// TIA Portal V20 export
FUNCTION "01 T5 EXCENTRIC Alarms" : Void   // FC1118, LAD
TITLE = ALARMS
{ S7_Optimized_Access := 'TRUE' }
// stored: AutoNumber false, IsIECCheckEnabled true, SetENOAutomatically false
   VAR_TEMP
      Trash : Bool;
   END_VAR
BEGIN

REGION Network 1: ============ ALARMS RESET ============
END_REGION

REGION Network 2: Alarms Reset
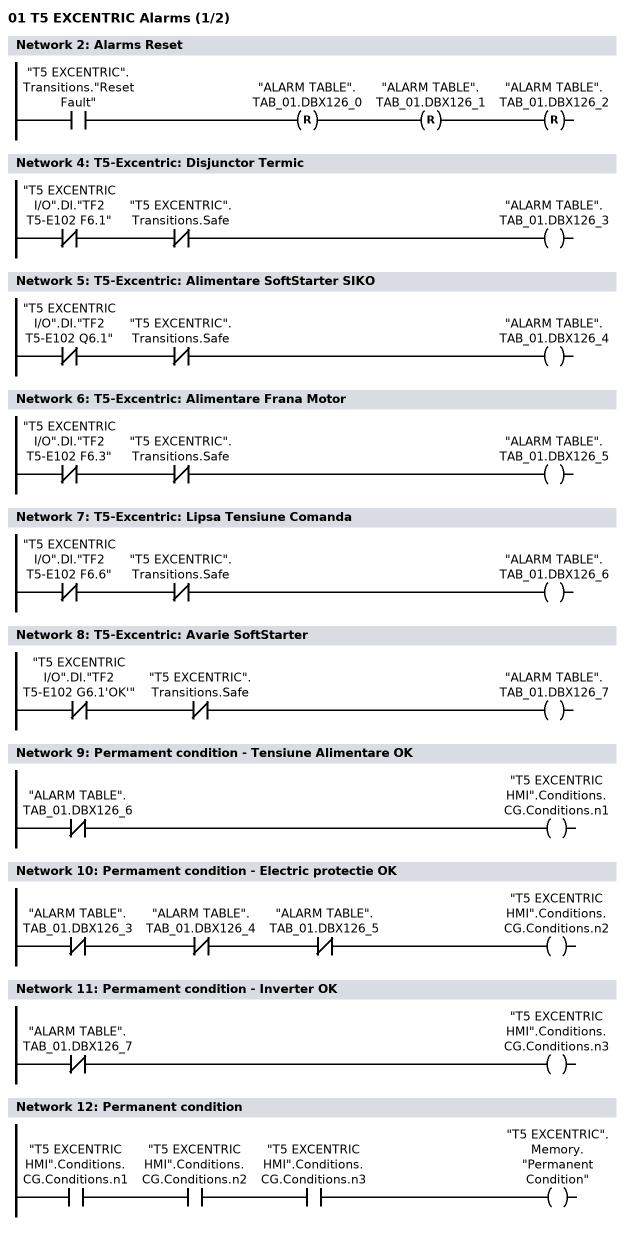
   RUNG wire#powerrail
      Contact( "T5 EXCENTRIC".Transitions."Reset Fault" )
      R_Coil( "ALARM TABLE".TAB_01.DBX126_0 )
      R_Coil( "ALARM TABLE".TAB_01.DBX126_1 )
      R_Coil( "ALARM TABLE".TAB_01.DBX126_2 )
   END_RUNG
   // the same network as SCL:
   IF "T5 EXCENTRIC".Transitions."Reset Fault" THEN
       "ALARM TABLE".TAB_01.DBX126_0 := FALSE;
       "ALARM TABLE".TAB_01.DBX126_1 := FALSE;
       "ALARM TABLE".TAB_01.DBX126_2 := FALSE;
   END_IF;
END_REGION

REGION Network 3: ============ PERMANENT CONDITIONS ============
END_REGION

REGION Network 4: T5-Excentric: Disjunctor Termic
   RUNG wire#powerrail
      I_Contact( "T5 EXCENTRIC I/O".DI."TF2 T5-E102 F6.1" )
      I_Contact( "T5 EXCENTRIC".Transitions.Safe )
      Coil( "ALARM TABLE".TAB_01.DBX126_3 )
   END_RUNG
   // the same network as SCL:
   "ALARM TABLE".TAB_01.DBX126_3 := NOT "T5 EXCENTRIC I/O".DI."TF2 T5-E102 F6.1" AND NOT "T5 EXCENTRIC".Transitions.Safe;
END_REGION

REGION Network 5: T5-Excentric: Alimentare SoftStarter SIKO
   RUNG wire#powerrail
      I_Contact( "T5 EXCENTRIC I/O".DI."TF2 T5-E102 Q6.1" )
      I_Contact( "T5 EXCENTRIC".Transitions.Safe )
      Coil( "ALARM TABLE".TAB_01.DBX126_4 )
   END_RUNG
   // the same network as SCL:
   "ALARM TABLE".TAB_01.DBX126_4 := NOT "T5 EXCENTRIC I/O".DI."TF2 T5-E102 Q6.1" AND NOT "T5 EXCENTRIC".Transitions.Safe;
END_REGION

REGION Network 6: T5-Excentric: Alimentare Frana Motor
   RUNG wire#powerrail
      I_Contact( "T5 EXCENTRIC I/O".DI."TF2 T5-E102 F6.3" )
      I_Contact( "T5 EXCENTRIC".Transitions.Safe )
      Coil( "ALARM TABLE".TAB_01.DBX126_5 )
   END_RUNG
   // the same network as SCL:
   "ALARM TABLE".TAB_01.DBX126_5 := NOT "T5 EXCENTRIC I/O".DI."TF2 T5-E102 F6.3" AND NOT "T5 EXCENTRIC".Transitions.Safe;
END_REGION

REGION Network 7: T5-Excentric: Lipsa Tensiune Comanda
   RUNG wire#powerrail
      I_Contact( "T5 EXCENTRIC I/O".DI."TF2 T5-E102 F6.6" )
      I_Contact( "T5 EXCENTRIC".Transitions.Safe )
      Coil( "ALARM TABLE".TAB_01.DBX126_6 )
   END_RUNG
   // the same network as SCL:
   "ALARM TABLE".TAB_01.DBX126_6 := NOT "T5 EXCENTRIC I/O".DI."TF2 T5-E102 F6.6" AND NOT "T5 EXCENTRIC".Transitions.Safe;
END_REGION

REGION Network 8: T5-Excentric: Avarie SoftStarter
   RUNG wire#powerrail
      I_Contact( "T5 EXCENTRIC I/O".DI."TF2 T5-E102 G6.1'OK'" )
      I_Contact( "T5 EXCENTRIC".Transitions.Safe )
      Coil( "ALARM TABLE".TAB_01.DBX126_7 )
   END_RUNG
   // the same network as SCL:
   "ALARM TABLE".TAB_01.DBX126_7 := NOT "T5 EXCENTRIC I/O".DI."TF2 T5-E102 G6.1'OK'" AND NOT "T5 EXCENTRIC".Transitions.Safe;
END_REGION

REGION Network 9: Permament condition - Tensiune Alimentare OK
   RUNG wire#powerrail
      I_Contact( "ALARM TABLE".TAB_01.DBX126_6 )
      Coil( "T5 EXCENTRIC HMI".Conditions.CG.Conditions.n1 )
   END_RUNG
   // the same network as SCL:
   "T5 EXCENTRIC HMI".Conditions.CG.Conditions.n1 := NOT "ALARM TABLE".TAB_01.DBX126_6;
END_REGION

REGION Network 10: Permament condition - Electric protectie OK
   RUNG wire#powerrail
      I_Contact( "ALARM TABLE".TAB_01.DBX126_3 )
      I_Contact( "ALARM TABLE".TAB_01.DBX126_4 )
      I_Contact( "ALARM TABLE".TAB_01.DBX126_5 )
      Coil( "T5 EXCENTRIC HMI".Conditions.CG.Conditions.n2 )
   END_RUNG
   // the same network as SCL:
   "T5 EXCENTRIC HMI".Conditions.CG.Conditions.n2 := NOT "ALARM TABLE".TAB_01.DBX126_3 AND NOT "ALARM TABLE".TAB_01.DBX126_4 AND NOT "ALARM TABLE".TAB_01.DBX126_5;
END_REGION

REGION Network 11: Permament condition - Inverter OK
   RUNG wire#powerrail
      I_Contact( "ALARM TABLE".TAB_01.DBX126_7 )
      Coil( "T5 EXCENTRIC HMI".Conditions.CG.Conditions.n3 )
   END_RUNG
   // the same network as SCL:
   "T5 EXCENTRIC HMI".Conditions.CG.Conditions.n3 := NOT "ALARM TABLE".TAB_01.DBX126_7;
END_REGION

REGION Network 12: Permanent condition
   RUNG wire#powerrail
      Contact( "T5 EXCENTRIC HMI".Conditions.CG.Conditions.n1 )
      Contact( "T5 EXCENTRIC HMI".Conditions.CG.Conditions.n2 )
      Contact( "T5 EXCENTRIC HMI".Conditions.CG.Conditions.n3 )
      Coil( "T5 EXCENTRIC".Memory."Permanent Condition" )
   END_RUNG
   // the same network as SCL:
   "T5 EXCENTRIC".Memory."Permanent Condition" := "T5 EXCENTRIC HMI".Conditions.CG.Conditions.n1 AND "T5 EXCENTRIC HMI".Conditions.CG.Conditions.n2 AND "T5 EXCENTRIC HMI".Conditions.CG.Conditions.n3;
END_REGION

REGION Network 13: ======= MACHINE MOVEMENT CONTROL (SENSORS / ENCODERS / INTERLOCKS) =======
END_REGION

REGION Network 14: T5-Excentric: TimeOut Deplasare 'Inainte'
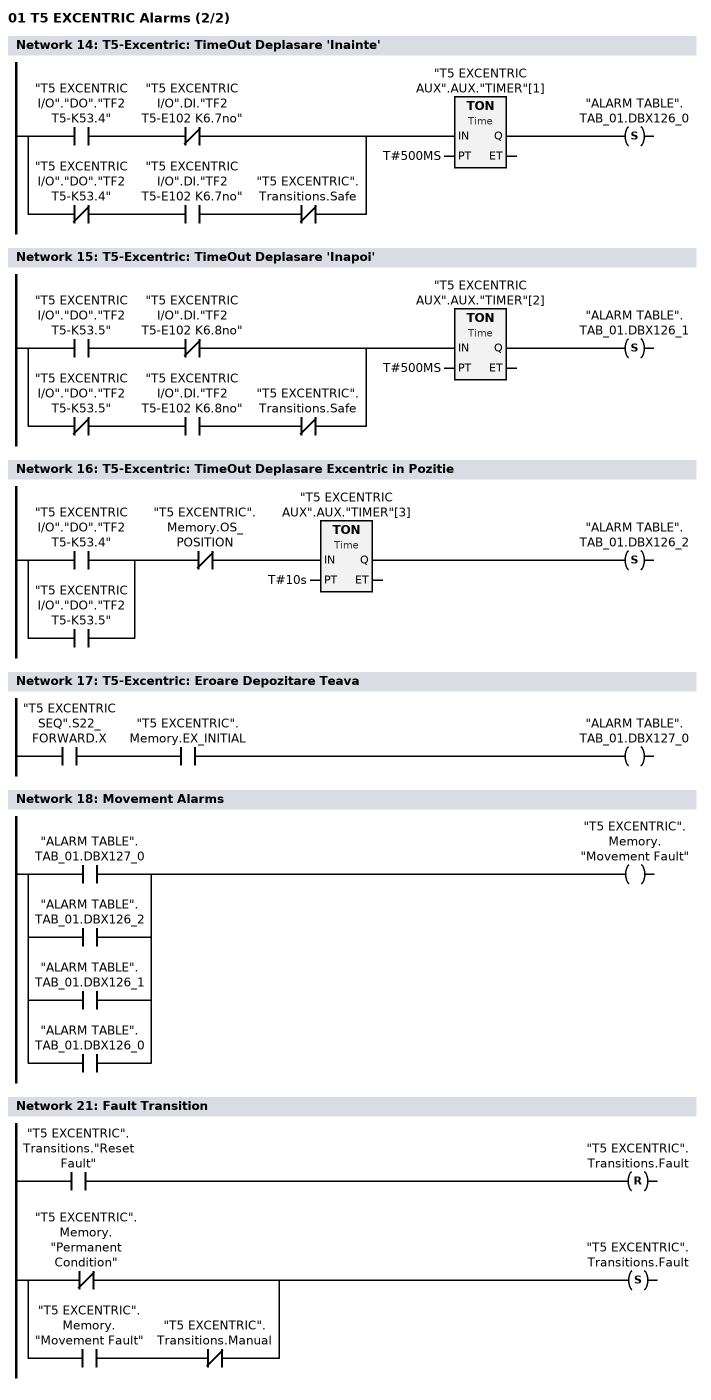
   RUNG wire#powerrail
      Contact( "T5 EXCENTRIC I/O"."DO"."TF2 T5-K53.4" )
      I_Contact( "T5 EXCENTRIC I/O".DI."TF2 T5-E102 K6.7no" )
      wire#w1
      { S7_Templates := "time_type := Time" } "T5 EXCENTRIC AUX".AUX."TIMER"[1].TON(pt := T#500MS, et =>)
      S_Coil( "ALARM TABLE".TAB_01.DBX126_0 )
   END_RUNG
   RUNG wire#powerrail
      I_Contact( "T5 EXCENTRIC I/O"."DO"."TF2 T5-K53.4" )
      Contact( "T5 EXCENTRIC I/O".DI."TF2 T5-E102 K6.7no" )
      I_Contact( "T5 EXCENTRIC".Transitions.Safe )
   END_RUNG wire#w1
   // the same network as SCL:
   "T5 EXCENTRIC AUX".AUX."TIMER"[1].TON(IN := ("T5 EXCENTRIC I/O"."DO"."TF2 T5-K53.4" AND NOT "T5 EXCENTRIC I/O".DI."TF2 T5-E102 K6.7no") OR (NOT "T5 EXCENTRIC I/O"."DO"."TF2 T5-K53.4" AND "T5 EXCENTRIC I/O".DI."TF2 T5-E102 K6.7no" AND NOT "T5 EXCENTRIC".Transitions.Safe),
                           PT := T#500MS);
   IF "T5 EXCENTRIC AUX".AUX."TIMER"[1].Q THEN "ALARM TABLE".TAB_01.DBX126_0 := TRUE; END_IF;
END_REGION

REGION Network 15: T5-Excentric: TimeOut Deplasare 'Inapoi'
   RUNG wire#powerrail
      Contact( "T5 EXCENTRIC I/O"."DO"."TF2 T5-K53.5" )
      I_Contact( "T5 EXCENTRIC I/O".DI."TF2 T5-E102 K6.8no" )
      wire#w1
      { S7_Templates := "time_type := Time" } "T5 EXCENTRIC AUX".AUX."TIMER"[2].TON(pt := T#500MS, et =>)
      S_Coil( "ALARM TABLE".TAB_01.DBX126_1 )
   END_RUNG
   RUNG wire#powerrail
      I_Contact( "T5 EXCENTRIC I/O"."DO"."TF2 T5-K53.5" )
      Contact( "T5 EXCENTRIC I/O".DI."TF2 T5-E102 K6.8no" )
      I_Contact( "T5 EXCENTRIC".Transitions.Safe )
   END_RUNG wire#w1
   // the same network as SCL:
   "T5 EXCENTRIC AUX".AUX."TIMER"[2].TON(IN := ("T5 EXCENTRIC I/O"."DO"."TF2 T5-K53.5" AND NOT "T5 EXCENTRIC I/O".DI."TF2 T5-E102 K6.8no") OR (NOT "T5 EXCENTRIC I/O"."DO"."TF2 T5-K53.5" AND "T5 EXCENTRIC I/O".DI."TF2 T5-E102 K6.8no" AND NOT "T5 EXCENTRIC".Transitions.Safe),
                           PT := T#500MS);
   IF "T5 EXCENTRIC AUX".AUX."TIMER"[2].Q THEN "ALARM TABLE".TAB_01.DBX126_1 := TRUE; END_IF;
END_REGION

REGION Network 16: T5-Excentric: TimeOut Deplasare Excentric in Pozitie
   RUNG wire#powerrail
      Contact( "T5 EXCENTRIC I/O"."DO"."TF2 T5-K53.4" )
      wire#w1
      I_Contact( "T5 EXCENTRIC".Memory.OS_POSITION )
      { S7_Templates := "time_type := Time" } "T5 EXCENTRIC AUX".AUX."TIMER"[3].TON(pt := T#10s, et =>)
      S_Coil( "ALARM TABLE".TAB_01.DBX126_2 )
   END_RUNG
   RUNG wire#powerrail
      Contact( "T5 EXCENTRIC I/O"."DO"."TF2 T5-K53.5" )
   END_RUNG wire#w1
   // the same network as SCL:
   "T5 EXCENTRIC AUX".AUX."TIMER"[3].TON(IN := ("T5 EXCENTRIC I/O"."DO"."TF2 T5-K53.4" OR "T5 EXCENTRIC I/O"."DO"."TF2 T5-K53.5") AND NOT "T5 EXCENTRIC".Memory.OS_POSITION,
                           PT := T#10s);
   IF "T5 EXCENTRIC AUX".AUX."TIMER"[3].Q THEN "ALARM TABLE".TAB_01.DBX126_2 := TRUE; END_IF;
END_REGION

REGION Network 17: T5-Excentric: Eroare Depozitare Teava
   RUNG wire#powerrail
      Contact( "T5 EXCENTRIC SEQ".S22_FORWARD.X )
      Contact( "T5 EXCENTRIC".Memory.EX_INITIAL )
      Coil( "ALARM TABLE".TAB_01.DBX127_0 )
   END_RUNG
   // the same network as SCL:
   "ALARM TABLE".TAB_01.DBX127_0 := "T5 EXCENTRIC SEQ".S22_FORWARD.X AND "T5 EXCENTRIC".Memory.EX_INITIAL;
END_REGION

REGION Network 18: Movement Alarms
   RUNG wire#powerrail
      Contact( "ALARM TABLE".TAB_01.DBX127_0 )
      wire#w1
      Coil( "T5 EXCENTRIC".Memory."Movement Fault" )
   END_RUNG
   RUNG wire#powerrail
      Contact( "ALARM TABLE".TAB_01.DBX126_2 )
   END_RUNG wire#w1
   RUNG wire#powerrail
      Contact( "ALARM TABLE".TAB_01.DBX126_1 )
   END_RUNG wire#w1
   RUNG wire#powerrail
      Contact( "ALARM TABLE".TAB_01.DBX126_0 )
   END_RUNG wire#w1
   // the same network as SCL:
   "T5 EXCENTRIC".Memory."Movement Fault" := "ALARM TABLE".TAB_01.DBX127_0 OR "ALARM TABLE".TAB_01.DBX126_2 OR "ALARM TABLE".TAB_01.DBX126_1 OR "ALARM TABLE".TAB_01.DBX126_0;
END_REGION

REGION Network 19: ======= OTHER ALARMS =======
END_REGION

REGION Network 20: ======= FAULT =======
END_REGION

REGION Network 21: Fault Transition
   RUNG wire#powerrail
      Contact( "T5 EXCENTRIC".Transitions."Reset Fault" )
      R_Coil( "T5 EXCENTRIC".Transitions.Fault )
   END_RUNG
   RUNG wire#powerrail
      I_Contact( "T5 EXCENTRIC".Memory."Permanent Condition" )
      wire#w1
      S_Coil( "T5 EXCENTRIC".Transitions.Fault )
   END_RUNG
   RUNG wire#powerrail
      Contact( "T5 EXCENTRIC".Memory."Movement Fault" )
      I_Contact( "T5 EXCENTRIC".Transitions.Manual )
   END_RUNG wire#w1
   // the same network as SCL:
   IF "T5 EXCENTRIC".Transitions."Reset Fault" THEN "T5 EXCENTRIC".Transitions.Fault := FALSE; END_IF;
   IF NOT "T5 EXCENTRIC".Memory."Permanent Condition" OR ("T5 EXCENTRIC".Memory."Movement Fault" AND NOT "T5 EXCENTRIC".Transitions.Manual) THEN
       "T5 EXCENTRIC".Transitions.Fault := TRUE;
   END_IF;
END_REGION
END_FUNCTION
